TYPE ST_ACDCCharger_Service :
STRUCT
END_STRUCT
END_TYPE

(* stored: Version 1.1.0.1, ProductVersion 3.1.4026.18
   DUT ST_ACDCCharger_Service: Id {421c01bf-48df-4106-b173-4f5705cbbd23} *)
